FUNCTION_BLOCK FB_ModeStateControl_Base
VAR_INPUT
	i_bReqAutomatic : BOOL;
	i_bReqManual : BOOL;
	i_bReqMaintenance : BOOL;
	i_bReqIoTest : BOOL;
	i_bReqCleaning : BOOL;	

	i_bReqStart : BOOL;
	i_bReqStop : BOOL;
	i_bReqReset : BOOL;
	i_bStaStopped : BOOL;
END_VAR
VAR_OUTPUT
END_VAR
VAR
	s_bInitDone : BOOL := FALSE;	

	s_eCtrlMode : E_CtrlMode := E_CtrlMode.IDLE;
	s_eCtrlState : E_CtrlState := E_CtrlState.STOPPED;	
END_VAR

METHOD PRIVATE _m_Init : BOOL

//Mode buttons
s_fbHmiBtnModeAutomatic.p_eButtontype := E_HmiButtonType.PUSHBUTTON;
s_fbHmiBtnModeAutomatic.p_bStaVisible := FALSE;
s_fbHmiBtnModeAutomatic.p_bStaEnabled := FALSE;
s_fbHmiBtnModeAutomatic.p_sBtnText := 'Automatic';

s_fbHmiBtnModeManual.p_eButtontype := E_HmiButtonType.PUSHBUTTON;
s_fbHmiBtnModeManual.p_bStaVisible := FALSE;
s_fbHmiBtnModeManual.p_bStaEnabled := FALSE;
s_fbHmiBtnModeManual.p_sBtnText := 'Manual';

s_fbHmiBtnModeMaintenance.p_eButtontype := E_HmiButtonType.PUSHBUTTON;
s_fbHmiBtnModeMaintenance.p_bStaVisible := FALSE;
s_fbHmiBtnModeMaintenance.p_bStaEnabled := FALSE;
s_fbHmiBtnModeMaintenance.p_sBtnText := 'Maintenance';

s_fbHmiBtnModeIO.p_eButtontype := E_HmiButtonType.PUSHBUTTON;
s_fbHmiBtnModeIO.p_bStaVisible := FALSE;
s_fbHmiBtnModeIO.p_bStaEnabled := FALSE;
s_fbHmiBtnModeIO.p_sBtnText := 'IO';

s_fbHmiBtnModeCleaning.p_eButtontype := E_HmiButtonType.PUSHBUTTON;
s_fbHmiBtnModeCleaning.p_bStaVisible := FALSE;
s_fbHmiBtnModeCleaning.p_bStaEnabled := FALSE;
s_fbHmiBtnModeCleaning.p_sBtnText := 'Cleaning';

//State buttons
s_fbHmiBtnStateStart.p_eButtontype := E_HmiButtonType.PUSHBUTTON;
s_fbHmiBtnStateStart.p_bStaVisible := FALSE;
s_fbHmiBtnStateStart.p_bStaEnabled := FALSE;
s_fbHmiBtnStateStart.p_sBtnText := 'Start';

s_fbHmiBtnStateStop.p_eButtontype := E_HmiButtonType.PUSHBUTTON;
s_fbHmiBtnStateStop.p_bStaVisible := FALSE;
s_fbHmiBtnStateStop.p_bStaEnabled := FALSE;
s_fbHmiBtnStateStop.p_sBtnText := 'Stop';

s_fbHmiBtnStateReset.p_eButtontype := E_HmiButtonType.PUSHBUTTON;
s_fbHmiBtnStateReset.p_bStaVisible := FALSE;
s_fbHmiBtnStateReset.p_bStaEnabled := FALSE;
s_fbHmiBtnStateReset.p_sBtnText := 'Reset';

_m_Init := TRUE;
END_METHOD

METHOD PUBLIC m_Main : BOOL

IF (s_eCtrlState = E_CtrlState.IDLE) OR (s_eCtrlState = E_CtrlState.STOPPED) THEN
	IF i_bReqAutomatic THEN
		s_eCtrlMode := E_CtrlMode.AUTOMATIC;
	ELSIF i_bReqManual THEN
		s_eCtrlMode := E_CtrlMode.MANUAL;
	ELSIF i_bReqMaintenance THEN
		s_eCtrlMode := E_CtrlMode.MAINTENANCE;
	ELSIF i_bReqIoTest THEN
		s_eCtrlMode := E_CtrlMode.IO;
	ELSIF i_bReqCleaning THEN
		s_eCtrlMode := E_CtrlMode.CLEANING;
	END_IF
END_IF

CASE s_eCtrlMode OF
	E_CtrlMode.IDLE:
		;//Nothing
	
	E_CtrlMode.AUTOMATIC:
		m_ModeAutomatic();
	
	E_CtrlMode.MANUAL:
		m_ModeManual();
	
	E_CtrlMode.MAINTENANCE:
		m_ModeMaintenance();
	
	E_CtrlMode.IO:
		m_ModeIoTest();
		
	E_CtrlMode.CLEANING:
		m_ModeCleaning();
		
	ELSE
		s_eCtrlMode := E_CtrlMode.IDLE;
END_CASE

CASE s_eCtrlState OF
	E_CtrlState.STOPPED:
		m_StateStopped();
		
		IF i_bReqReset THEN
			s_eCtrlState := E_CtrlState.IDLE;
		END_IF	
		
	E_CtrlState.IDLE:
		m_StateIdle();
		
		IF i_bReqStop THEN
			s_eCtrlState := E_CtrlState.STOPPING;
		ELSIF i_bReqStart THEN
			s_eCtrlState := E_CtrlState.RUNNING;
		END_IF
	
	E_CtrlState.RUNNING:
		m_StateRunning();
		
		IF i_bReqStop THEN
			s_eCtrlState := E_CtrlState.STOPPING;
		END_IF
			
	E_CtrlState.STOPPING:
		m_StateStopping();
		
		IF i_bStaStopped THEN
			s_eCtrlState := E_CtrlState.STOPPED;
		END_IF
	
	ELSE
		s_eCtrlState := E_CtrlState.STOPPED;
END_CASE

m_Main := TRUE;
END_METHOD

METHOD PUBLIC m_ModeAutomatic : BOOL
END_METHOD

METHOD PUBLIC m_ModeCleaning : BOOL
END_METHOD

METHOD PUBLIC m_ModeIoTest : BOOL
END_METHOD

METHOD PUBLIC m_ModeMaintenance : BOOL
END_METHOD

METHOD PUBLIC m_ModeManual : BOOL
END_METHOD

METHOD PUBLIC m_StateIdle : BOOL
END_METHOD

METHOD PUBLIC m_StateRunning : BOOL
END_METHOD

METHOD PUBLIC m_StateStopped : BOOL
END_METHOD

METHOD PUBLIC m_StateStopping : BOOL
END_METHOD

END_FUNCTION_BLOCK

(* stored: Version 1.1.0.1, ProductVersion 3.1.4024.12
   POU FB_ModeStateControl_Base: Id {0ff31c57-5f64-4e23-ba53-7c57d2a6b21a}, SpecialFunc None
   Method _m_Init: Id {0019b3fd-c704-42a7-8153-90eb9278931b}
   Method m_Main: Id {6c552307-b2a4-4386-9ac6-29f707c1b3c2}
   Method m_ModeAutomatic: Id {e990f1a2-dbac-46ab-b9fa-3e2db4742949}
   Method m_ModeCleaning: Id {719eef6e-a547-4145-9820-6ac1e3772c8e}
   Method m_ModeIoTest: Id {3d73adce-d293-4a9c-aec0-9275c0db02ef}
   Method m_ModeMaintenance: Id {5b5130cb-51aa-4e7e-8d5a-a00d3d24864e}
   Method m_ModeManual: Id {daaee783-e776-4c37-b94c-4e2b57285428}
   Method m_StateIdle: Id {94e0b4c9-9c7b-4fe3-b7d8-03530dc9f43b}
   Method m_StateRunning: Id {4ddb2b3b-e0d3-40a1-b13b-038664c09471}
   Method m_StateStopped: Id {0f7c6642-355d-43b8-b178-611a57e55b50}
   Method m_StateStopping: Id {736b5d08-289d-4576-842e-2ffba08064f4} *)
